PROGRAM MAIN
VAR
	m : INT;
END_VAR

m := m + 1;

PrgMqttCom();

END_PROGRAM

(* stored: Version 1.1.0.1, ProductVersion 3.1.4020.12
   POU MAIN: Id {cc69c161-152a-42d3-b915-bdc8cc2f5bde}, SpecialFunc None *)
